// TwinCAT 3 PLC project PLC1
// ProjectVersion: 3.1.4024.0
// project tree:
//   DUTs/ E_FillState.TcDUT
//   GVLs/ GVL_Machine.TcGVL
//   POUs/ FB_Filler.TcPOU, FB_Homing.TcPOU, MAIN.TcPOU

// ---- DUTs/E_FillState.TcDUT
TYPE E_FillState :
(
    Idle   := 0,
    Dosing := 10,
    Done   := 20,
    Fault  := 99
) INT;
END_TYPE

// ---- GVLs/GVL_Machine.TcGVL
{attribute 'qualified_only'}
VAR_GLOBAL
    xRunRequest     : BOOL;
    xHomeSensor     : BOOL;
    xProductPresent : BOOL;
    rTargetVolume   : LREAL := 250.0;   // ml
END_VAR

// ---- POUs/FB_Filler.TcPOU
FUNCTION_BLOCK FB_Filler
VAR_INPUT
    ixStart          : BOOL;
    ixProductPresent : BOOL;
    irTargetVolume   : LREAL;   // ml
END_VAR
VAR_OUTPUT
    qxFilling  : BOOL;
    qxDone     : BOOL;
    qxError    : BOOL;
    qnErrorID  : UDINT;
END_VAR
VAR
    eState         : E_FillState;
    rActualVolume  : LREAL;     // ml
    fbDoseTimer    : TON;
END_VAR

CASE eState OF
    E_FillState.Idle:
        IF ixStart AND ixProductPresent THEN
            eState := E_FillState.Dosing;
        END_IF

    E_FillState.Dosing:
        qxFilling := TRUE;
        IF THIS^.DoseComplete() THEN
            eState := E_FillState.Done;
        END_IF

    E_FillState.Done:
        qxFilling := FALSE;
        qxDone := TRUE;
        IF NOT ixStart THEN
            eState := E_FillState.Idle;
        END_IF

    E_FillState.Fault:
        qxFilling := FALSE;
        qxError := TRUE;
        IF NOT ixStart THEN
            qxError := FALSE;
            eState := E_FillState.Idle;
        END_IF
ELSE
    eState := E_FillState.Fault;
END_CASE

METHOD DoseComplete : BOOL
VAR
    nSettleCount : DINT;
END_VAR
// Let the dose settle before comparing against the target.
WHILE fbDoseTimer.Q = FALSE DO
    nSettleCount := nSettleCount + 1;
    fbDoseTimer(IN := TRUE, PT := 250);
END_WHILE

IF rActualVolume = irTargetVolume THEN
    DoseComplete := TRUE;
END_IF
END_METHOD

END_FUNCTION_BLOCK

// ---- POUs/FB_Homing.TcPOU
FUNCTION_BLOCK FB_Homing
VAR_INPUT
    ixStart      : BOOL;
    ixHomeSensor : BOOL;
END_VAR
VAR_OUTPUT
    qxHomed : BOOL;
    qxError : BOOL;
END_VAR
VAR
    nStep : INT;
END_VAR

CASE nStep OF
    0:  // idle
        IF ixStart THEN
            nStep := 10;
        END_IF

    10: // driving to the home sensor, waiting for it to make
        IF ixHomeSensor THEN
            qxHomed := TRUE;
            nStep := 20;
        END_IF

    20: // homed, hold until the request drops
        IF NOT ixStart THEN
            qxHomed := FALSE;
            nStep := 0;
        END_IF

    99: // fault
        qxError := TRUE;
        IF NOT ixStart THEN
            qxError := FALSE;
            nStep := 0;
        END_IF
ELSE
    nStep := 99;
END_CASE

END_FUNCTION_BLOCK

// ---- POUs/MAIN.TcPOU
PROGRAM MAIN
VAR
    fbHoming : FB_Homing;
    fbFiller : FB_Filler;
END_VAR

fbHoming(ixStart := GVL_Machine.xRunRequest,
         ixHomeSensor := GVL_Machine.xHomeSensor);

fbFiller(ixStart := GVL_Machine.xRunRequest AND fbHoming.qxHomed,
         ixProductPresent := GVL_Machine.xProductPresent,
         irTargetVolume := GVL_Machine.rTargetVolume);

END_PROGRAM
